SUBAPPLICATION Uebung_020f2_AX (* DigitalInput_I1 auf DigitalOutput_Q1; AX_FB_TP; Impulsformend *)
  (* Standard: 61499-2; Description: Copyright (c) 2023 Meisterschulen am Ostbahnhof This program and the accompanying materials are made available under the terms of the Eclipse Public License 2.0 which is available at https://www.eclipse.org/legal/epl-2.0/ SPDX-License-Identifier: EPL-2.0 *)
  (* Version 1.0, 2023-10-23, Franz Höpfinger, Meisterschulen am Ostbahnhof, initial API and implementation and/or initial documentation *)
  PACKAGE Uebungen;
  IMPORT logiBUS::io::DI::logiBUS_DI::Input_I1;
  IMPORT logiBUS::io::DQ::logiBUS_DO::Output_Q1;
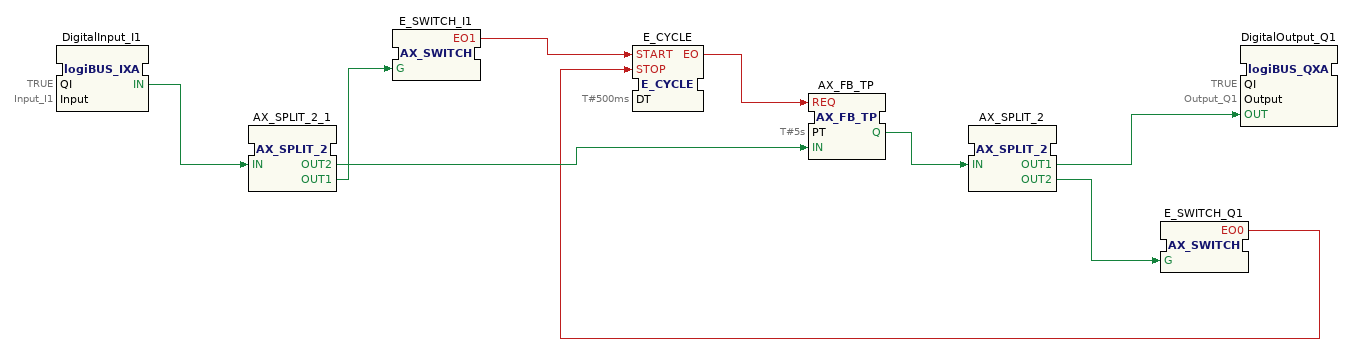
  (* E_CYCLE bestimmt, wie oft AX_FB_TP den ET aktualisert *)
  FBS
    E_SWITCH_I1 : adapter::events::unidirectional::AX_SWITCH;
    E_SWITCH_Q1 : adapter::events::unidirectional::AX_SWITCH;
    DigitalInput_I1 : logiBUS::io::DI::logiBUS_IXA(QI := TRUE, Input := Input_I1);
    AX_FB_TP : adapter::iec61131::timers::AX_FB_TP(PT := T#5s);
    DigitalOutput_Q1 : logiBUS::io::DQ::logiBUS_QXA(QI := TRUE, Output := Output_Q1);
    E_CYCLE : iec61499::events::E_CYCLE(DT := T#500ms);
    AX_SPLIT_2 : adapter::events::unidirectional::AX_SPLIT_2;
    AX_SPLIT_2_1 : adapter::events::unidirectional::AX_SPLIT_2;
  END_FBS
  EVENT_CONNECTIONS
    E_SWITCH_I1.EO1 TO E_CYCLE.START;
    E_SWITCH_Q1.EO0 TO E_CYCLE.STOP;
    E_CYCLE.EO TO AX_FB_TP.REQ;
  END_CONNECTIONS
  ADAPTER_CONNECTIONS
    AX_SPLIT_2_1.OUT2 TO AX_FB_TP.IN;
    AX_FB_TP.Q TO AX_SPLIT_2.IN;
    AX_SPLIT_2.OUT1 TO DigitalOutput_Q1.OUT;
    AX_SPLIT_2.OUT2 TO E_SWITCH_Q1.G;
    AX_SPLIT_2_1.OUT1 TO E_SWITCH_I1.G;
    DigitalInput_I1.IN TO AX_SPLIT_2_1.IN;
  END_CONNECTIONS
END_SUBAPPLICATION
